{attribute 'pack_mode' := '1'}
TYPE T_PtpDiag : // Holds the data from the PTP Diag section of the EL6688 CoE items
STRUCT
	numMembers: UINT;  // Added by FB_EcCoESdoReadEx.
	PTPVersion: UINT;
	PTPState: UINT;
	ClockIdentity: ARRAY[0..7] OF BYTE;
	ParentPortIdentity: ARRAY[0..9] OF BYTE;
	GramdmasterIdentity: ARRAY [0..7] OF BYTE;
	OffsetFromMaster: DINT;
	MeanPathDelay:UDINT;
	StepsRemoved: UINT;
	SyncSequece: UINT;
	Timescale: UINT;
	CurrentUtcOffset: INT;
	CurrentUtcOffsetIsValid: UINT;
	Leap61: UINT;
	Leap59: UINT;
	EpochNumber: UINT;
END_STRUCT
END_TYPE

(* stored: Version 1.1.0.1, ProductVersion 3.1.4022.18
   DUT T_PtpDiag: Id {913bc9c7-bb8b-4f1f-acd3-92d64244d25d} *)
